PROGRAM PRG_TESTS
VAR
    fbTestSuite1Instance1 : FB_TestSuite1;
END_VAR

TcUnit.RUN();

END_PROGRAM

(* stored: Version 1.1.0.1, ProductVersion 3.1.4024.12
   POU PRG_TESTS: Id {2f8fcc6e-c36b-40b5-a0ea-8b06b18e1a90}, SpecialFunc None *)
